FUNCTION_BLOCK DSCYL_MDL (* Model for a Double-Stroke Cylinder, Externally Clocked *)
  (* Standard: 61499-1 *)
  (* Version 0.2, 2008-06-27, JHC, Holobloc Inc, Adapted to modified WTAV_UINT interface (IN1/IN2 replace X1/X2). *)
  (* Version 0.1, 2005-06-01, JHC, Holobloc Inc, Re-compiled with new emitter. *)
  (* Version 0.0, 2003-03-17, JHC, Rockwell Automation, Adapted from old DSCYL_MV. *)
  (* Compiler header: package fb.rt.mach; import fb.rt.math.*; import fb.rt.mva.*; *)
  (* Compiler Java Sun JDK 1.4.2 *)
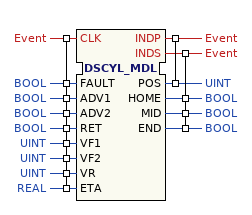
  EVENT_INPUT
    CLK WITH FAULT, ADV1, ADV2, RET, VF1, VF2, VR, ETA; (* External Clock Event *)
  END_EVENT
  EVENT_OUTPUT
    INDP WITH POS; (* Position Change Indication *)
    INDS WITH HOME, MID, END; (* Sensor Change Indication *)
  END_EVENT
  VAR_INPUT
    FAULT : BOOL; (* 0=Enable,1=Simulate Fault *)
    ADV1 : BOOL; (* ADVANCE Cyl#1 *)
    ADV2 : BOOL; (* ADVANCE Cyl#2 *)
    RET : BOOL; (* RETRACT Both Cylinders *)
    VF1 : UINT; (* Cyl#1 ADVANCE speed in %FS per CLK event *)
    VF2 : UINT; (* Cyl#2 ADVANCE speed in %FS per CLK event *)
    VR : UINT; (* RETRACT speed in %FS per CLK event *)
    ETA : REAL := 0.5; (* Length ratio:Cyl#1/(Cyl#1+Cyl#2) *)
  END_VAR
  VAR_OUTPUT
    POS : UINT; (* End effector position *)
    HOME : BOOL; (* Both cylinders HOME *)
    MID : BOOL; (* CYL1 at END,CYL2 HOME *)
    END : BOOL; (* Both cylinders at END *)
  END_VAR
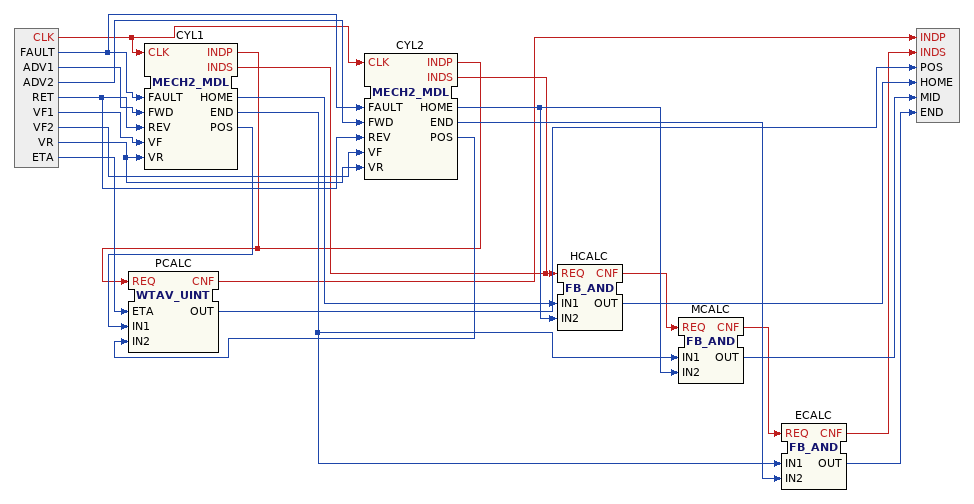
  FBS
    CYL1 : MECH2_MDL;
    CYL2 : MECH2_MDL;
    PCALC : WTAV_UINT;
    HCALC : FB_AND;
    MCALC : FB_AND;
    ECALC : FB_AND;
  END_FBS
  EVENT_CONNECTIONS
    HCALC.CNF TO MCALC.REQ;
    MCALC.CNF TO ECALC.REQ;
    CYL1.INDP TO PCALC.REQ;
    CYL2.INDP TO PCALC.REQ;
    PCALC.CNF TO INDP;
    CYL1.INDS TO HCALC.REQ;
    CYL2.INDS TO HCALC.REQ;
    ECALC.CNF TO INDS;
    CLK TO CYL1.CLK;
    CLK TO CYL2.CLK;
  END_CONNECTIONS
  DATA_CONNECTIONS
    FAULT TO CYL1.FAULT;
    FAULT TO CYL2.FAULT;
    ADV1 TO CYL1.FWD;
    ADV2 TO CYL2.FWD;
    RET TO CYL1.REV;
    RET TO CYL2.REV;
    ETA TO PCALC.ETA;
    CYL1.HOME TO HCALC.IN1;
    CYL2.HOME TO HCALC.IN2;
    CYL1.END TO MCALC.IN1;
    CYL2.HOME TO MCALC.IN2;
    CYL1.END TO ECALC.IN1;
    CYL2.END TO ECALC.IN2;
    CYL1.POS TO PCALC.IN1;
    CYL2.POS TO PCALC.IN2;
    HCALC.OUT TO HOME;
    MCALC.OUT TO MID;
    ECALC.OUT TO END;
    PCALC.OUT TO POS;
    VF1 TO CYL1.VF;
    VR TO CYL1.VR;
    VF2 TO CYL2.VF;
    VR TO CYL2.VR;
  END_CONNECTIONS
END_FUNCTION_BLOCK
